{attribute addProperty BoxType "EL9110-0000-0016"}
{attribute addProperty Id "PowerOKAT %I*PowerOK_E4AEF59E810WcStateAT %I*WcState_F855686C1620InfoDataAT %I*InfoData_192954DE1620"}
{attribute addProperty CRC "3601765323"}
{attribute addProperty SizeInBites "40"}
{attribute addProperty SizeInBytes "5"}
TYPE EL9110_CB6430E0 :
STRUCT
	{attribute addProperty Name "PowerOK"}
	PowerOK : PowerOK_E4AEF59E;
	{attribute addProperty Name "WcState"}
	WcState : WcState_F855686C;
	{attribute addProperty Name "InfoData"}
	InfoData : InfoData_192954DE;
END_STRUCT
END_TYPE

(* stored: Version 1.2.0.0, ProductVersion 3.1.4024.9
   DUT EL9110_CB6430E0: Id {d2eb532b-f1cf-46c9-9307-2e3c723ee15b} *)
